# EPICS IOC start-up script: iocsh/LakeShore_330.iocsh
# ### LakeShore_330.iocsh ###

#- ###################################################
#- PREFIX         - IOC Prefix
#- INSTANCE       - Instance Prefix
#- PORT           - Serial port name
#- IP             - Location of IP module
#- ###################################################

iocshLoad("$(IP)/iocsh/setSerialParams.iocsh", "BAUD=1200, BITS=7, STOP=1, PARITY=odd")

asynOctetSetInputEos( "$(PORT)", -1, "\r")
asynOctetSetOutputEos("$(PORT)", -1, "\n")

dbLoadRecords("$(IP)/ipApp/Db/LakeShore330.db", "P=$(PREFIX),Q=$(INSTANCE),PORT=$(PORT)")
